// TwinCAT 3 PLC project TcpIpServer_Ex1
// ProgramVersion: 3.1.4023.0
// libraries:
//   Tc2_Standard, * (Beckhoff Automation GmbH)
//   Tc2_System, * (Beckhoff Automation GmbH)
//   Tc2_TcpIp, * (Beckhoff Automation GmbH)
//   Tc2_Utilities, * (Beckhoff Automation GmbH)
//   Tc3_Module, * (Beckhoff Automation GmbH)
// project tree:
//   / PlcTask.TcTTO
//   POUs/ F_Resp.TcPOU, MAIN.TcPOU
// real-time tasks:
//   TASK PlcTask: cycle T#10ms, priority 20, ADS port 350

CONFIGURATION TcpIpServer_Ex1
    RESOURCE PLC ON TwinCAT3
        TASK PlcTask(INTERVAL := T#10ms, PRIORITY := 20);
        PROGRAM MAIN WITH PlcTask : MAIN;
    END_RESOURCE
END_CONFIGURATION

// ---- POUs/MAIN.TcPOU
PROGRAM MAIN
VAR
	xIsInit: BOOL;
	sLocalHost: STRING := '127.0.0.1';
	hServer: T_HSERVER;
	fbServer: FB_ServerClientConnection;
	fbSocketReceive: FB_SocketReceive;
	sData: STRING(255);
	nRec: INT;
	xRecData: BOOL;
	cNewRecData: INT;
	nLastError: UDINT;
	cRecError: INT;
	WaitNewReadTON: TON;
	nInvalidCase: INT;
	nBadCase: INT;
	sLastData: STRING(1000);
	startupWaitTON: TON;
	fbSocketCloseAll: FB_SocketCloseAll;
	fbSocketSend: FB_SocketSend;
	sSendString: STRING(1000) := 'Hello World';
	xSendString: BOOL;
	hres: INT;
END_VAR


	/// here is were we populate response string to any received message
sSendString := F_Resp() ; 

startupWaitTON( IN := NOT xIsInit, PT := T#5S ) ; 


IF NOT xIsInit AND startupWaitTON.Q THEN
	xIsInit := F_CreateServerHnd(
							sSrvNetID:= '' , 
							sLocalHost:= sLocalHost , 
							nLocalPort:= 1234 , 
							nMode:= LISTEN_MODE_CLOSEALL + CONNECT_MODE_ENABLEDBG , 
							bEnable:= FALSE , 
							hServer:= hServer ) ;
END_IF

fbSocketCloseAll(
	sSrvNetId:= , 
	bExecute:= NOT xIsInit , 
	tTimeout:= , 
	bBusy=> , 
	bError=> , 
	nErrId=> );

fbServer(
	hServer:= hServer , 
	eMode:=  , 
	sRemoteHost:= , 
	nRemotePort:= , 
	bEnable:= xIsInit , 
	tReconnect:= T#10S , 
	bBusy=> , 
	bError=> , 
	nErrID=> , 
	hSocket=> , 
	eState=> );
	
fbServer.eState ; 

CASE nRec OF
0: // wait for connected
	IF fbServer.eState = E_SOCKETCONNECTIONSTATE.eSOCKET_CONNECTED THEN
		//clear trigger bit
		xRecData := FALSE ; 
		//we are connected so we can try receiving data
		nRec := 10 ; 
	END_IF
10: // trigger receive check
	xRecData := TRUE ; 
	nRec := 20 ; 
20: // wait receive check complete
	IF NOT fbSocketReceive.bBusy THEN
		xRecData := FALSE ; 
		// check for not error
		IF NOT fbSocketReceive.bError THEN
			// check if data was received 
			IF fbSocketReceive.nRecBytes>0 THEN
				//we have new data, do something with it
				//...
				xSendString := TRUE ; 
				//latch last good data
				sLastData := sData ; 
				
				// we'll just increment a counter here
				cNewRecData := cNewRecData + 1; 
			ELSE
				// no new data. that's ok, we'll poll again in a little bit
				;
			END_IF
		ELSE
			// error on receive. latch last error
			nLastError := fbSocketReceive.nErrId ;
			// count receive errors 
			cRecError := cRecError + 1 ;
			xIsInit := FALSE ;  
		END_IF
		
		// any time we are done with polling for new data (good or fault)
		// we will wait some time before polling again
		nRec := 30 ; 
	END_IF
30:// wait to poll again
	WaitNewReadTON( IN := TRUE, PT := T#100MS ) ; 
	IF WaitNewReadTON.Q THEN
		//reset timer
		WaitNewReadTON( IN := FALSE ) ;
		xSendString := FALSE ;
		// if we are done waiting, then go back to case 0 and decide if ready to poll again
		nRec := 0 ; 
	END_IF
ELSE
	//always have an else case!
	//latch invalid internal state
	nInvalidCase := nRec ; 
	//count num of time in invalid case
	nBadCase := nBadCase + 1; 
	//go to init
	nRec := 0 ; 
END_CASE

fbSocketReceive(
	sSrvNetId:= , 
	hSocket:= fbServer.hSocket , 
	cbLen:= SIZEOF(sData) , 
	pDest:= ADR(sData) , 
	bExecute:= xRecData , 
	tTimeout:= , 
	bBusy=> , 
	bError=> , 
	nErrId=> , 
	nRecBytes=> );

	
fbSocketSend(
	sSrvNetId:= , 
	hSocket:= fbServer.hSocket , 
	cbLen:= LEN2(ADR(sSendString)) , 
	pSrc:= ADR(sSendString) , 
	bExecute:= xSendString , 
	tTimeout:= , 
	bBusy=> , 
	bError=> , 
	nErrId=> );
	
	
hres := len('{"header":{"status":0,"message":"Ok"},"data":{"LocState":2}}') ;

END_PROGRAM

// ---- POUs/F_Resp.TcPOU
FUNCTION F_Resp : STRING(1000)
VAR_INPUT
END_VAR
VAR
END_VAR

(*F_Resp := 'HTTP/1.1 200 OK
Pragma: no-cache
Cache-Control: no-cache
Content-Type: application/json
Content-Length: 000000000060

{"header":{"status":0,"message":"Ok"},"data":{"LocState":2}}' ; 

F_Resp :='HTTP/1.1 200 OK
Date: Mon, 13 Sep 2021 15:30:54 GMT
Content-Type: application/json; charset=utf-8
Content-Length: 306
Connection: close
ETag: W/"132-GAnpLnU3NsyDWLw+Gf+eTxqCEf4"
Vary: Accept-Encoding
set-cookie: sails.sid=s%3ARbq3Ifbyb8AiuNjiVzrtP_NHB-sZvxYf.9zLKJDJ4D%2BqNBmZaMIbFWYismpi%2FcQFMepKgrCN340s; Path=/; HttpOnly

{"args":{"foo1":"bar1","foo2":"bar2"},"headers":{"x-forwarded-proto":"http","x-forwarded-port":"80","host":"postman-echo.com","x-amzn-trace-id":"Root=1-613f6eae-285d2c4318f5ed6e1bf9ef23","user-agent":"TcHttpClient","accept-encoding":"gzip, deflate"},"url":"http://postman-echo.com/get?foo1=bar1&foo2=bar2"}';



F_Resp := 'HTTP/1.1 200 OK
Pragma: no-cache
Cache-Control: no-cache
Content-Type: application/json
Content-Length: 60

{"header":{"status":1,"message":"Ok"},"data":{"LocState":5}}' ;
*)

F_Resp := '{"status":0,"message":"Ok"},"data":{"LocState":2}';

END_FUNCTION
